FUNCTION xnrm2_l : LREAL
VAR_INPUT
    b_n: DINT;
    x: ARRAY [0..4] OF LREAL;
    ix0: DINT;
END_VAR
VAR
    scale: LREAL;
    kend: DINT;
    absxk: LREAL;
    t: LREAL;
    k: DINT;
END_VAR

xnrm2_l := 0.0;
IF b_n >= 1 THEN 
    IF b_n = 1 THEN 
        xnrm2_l := ABS(x[ix0 - 1]);
    ELSE 
        scale := 3.3121686421112381E-170;
        kend := (ix0 + b_n) - 1;
        k := ix0;
        WHILE k <= kend DO
            absxk := ABS(x[k - 1]);
            IF absxk > scale THEN 
                t := scale / absxk;
                xnrm2_l := ((xnrm2_l * t) * t) + 1.0;
                scale := absxk;
            ELSE 
                t := absxk / scale;
                xnrm2_l := (t * t) + xnrm2_l;
            END_IF;
            k := k + 1;
        END_WHILE;
        xnrm2_l := scale * SQRT(xnrm2_l);
    END_IF;
END_IF;

END_FUNCTION

(* stored: Version 1.1.0.1, ProductVersion 3.1.4024.12
   POU xnrm2_l: Id {9fef4206-4cf0-41d5-924c-ea67846627c7}, SpecialFunc None *)
